// TIA Portal V20 export
DATA_BLOCK "TimerTimeE001_DB"   // DB100
// stored: InstanceOfName TimerTime, InstanceOfType FB
"TimerTime"
   // VAR_INPUT
   //    TimeSP : Real;
   //    SafeTime : Bool;
   //    State : DWord;
   // END_VAR
   // VAR_OUTPUT
   //    TimerTime : DInt;
   // END_VAR
   // VAR
   //    TimeSafe : DInt;
   //    safed : Bool;
   // END_VAR
BEGIN
END_DATA_BLOCK
